SUBAPPLICATION SoftKeyT_PC_B_OPC_Adapter (* Geraet B (Station 12, 192.168.1.12): wie Toggle_RPC_FROM_Remote_QXA_OPC, aber CLIENT_0/SERVER_0-Trigger und AX_CLIENT_1_0 sind hinter EINEM AE_AX_SERVER_0_CLIENT_1_0-Baustein hinter einem einzigen bidirektionalen Adapter-Anschluss gebuendelt; AE_AX_AX_SPLIT speist sowohl DigitalOutput_Q1 als auch die Toggle-Flipflop-Logik (AE_AX_T_FF) - 'SUB style': das Protokoll steckt im MyLib::sys-Composite, nicht in der Resource des Geraets *)
  (* Standard: 61499-2; Description: Copyright (c) 2026 Meisterschulen am Ostbahnhof This program and the accompanying materials are made available under the terms of the Eclipse Public License 2.0 which is available at https://www.eclipse.org/legal/epl-2.0/ SPDX-License-Identifier: EPL-2.0 *)
  (* Version 1.0, 2026-09-04, Franz Höpfinger, Meisterschulen am Ostbahnhof, initial API and implementation and/or initial documentation *)
  PACKAGE MyLib::sys;
  IMPORT logiBUS::io::DQ::logiBUS_DO;
  IMPORT logiBUS::io::DQ::logiBUS_DO_S;
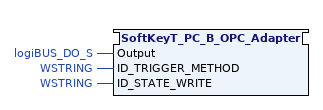
  VAR_INPUT
    Output : logiBUS::io::DQ::logiBUS_DO_S := logiBUS_DO::Invalid; (* Identify the Output Output_Q1..Q8 *)
    ID_TRIGGER_METHOD : WSTRING; (* Lokale Methodenadresse (ACTION=CREATE_METHOD) fuer den argumentlosen Trigger-Methodenaufruf, wird von Geraet A per CALL_METHOD aufgerufen *)
    ID_STATE_WRITE : WSTRING; (* Remote-Ziel-Adresse (BOOL, ACTION=WRITE) fuer den Flipflop-Zustand auf Geraet A *)
  END_VAR
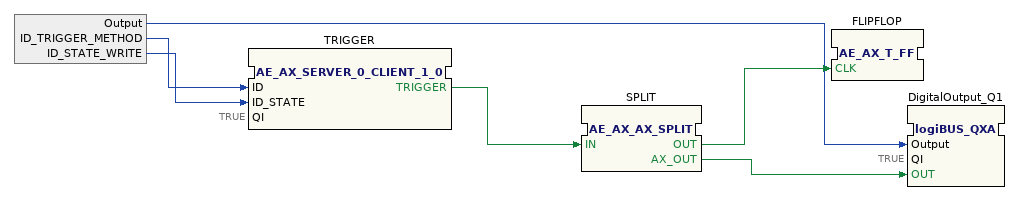
  FBS
    TRIGGER : adapter::net::AE_AX_SERVER_0_CLIENT_1_0(QI := TRUE);
    SPLIT : adapter::events::bidirectional::AE_AX_AX_SPLIT;
    FLIPFLOP : adapter::events::bidirectional::AE_AX_T_FF;
    DigitalOutput_Q1 : logiBUS::io::DQ::logiBUS_QXA(QI := TRUE);
  END_FBS
  DATA_CONNECTIONS
    Output TO DigitalOutput_Q1.Output;
    ID_TRIGGER_METHOD TO TRIGGER.ID;
    ID_STATE_WRITE TO TRIGGER.ID_STATE;
  END_CONNECTIONS
  ADAPTER_CONNECTIONS
    TRIGGER.TRIGGER TO SPLIT.IN;
    SPLIT.OUT TO FLIPFLOP.CLK;
    SPLIT.AX_OUT TO DigitalOutput_Q1.OUT;
  END_CONNECTIONS
END_SUBAPPLICATION
